Staubli VAL3: getObjectData.pgx

public program getObjectData(trsf& x_trObject[] (dimensions=1), num& x_nError[] (dimensions=1))
  local point l_pPoint
begin
  // This program returns the coordinates of the object
  // that have been pushed into the buffer by the detection lib.
  // This function is usefull when an advanced detection device
  // (e.g vision system) is in use.
  //
  // Input Param
  //  none
  //
  // Output Param
  //  x_trObject  : coordinates of the object
  //  x_nError    : Error code
  //    0 : No error
  //    1 : No data available
  //
  // Created 25-01-06                                   C.CURRIVAND
  //----------------------------------------------------------------
  //
  x_nError=0
  if nNumbOfUser[nIdxPull]!=0
    x_trObject=trDetectedCoord[nIdxPull]
  else
    //* No Object requested
    x_nError=1
    if cfg:bLog==true
      nErrVal[0]=nIdxPull
      call ut:addNumToString(sConvNum+"(getObjectData)>>"+sErrMsgList[x_nError],sMsg,"*",nErrVal)
      logMsg(sMsg)
    endIf
  endIf
end
